{attribute 'qualified_only'}
{attribute 'strict'}
TYPE AuftragsStatus :
(
	scan,
	start,
	end,
	vorwahl
);
END_TYPE

(* stored: Version 1.1.0.1, ProductVersion 3.1.4024.12
   DUT AuftragsStatus: Id {4e846d94-e9d7-49b0-b7ea-d0385d391a80} *)
